{attribute addProperty BoxType "EL1259-0000-0018"}
{attribute addProperty Id "StatusAT %I*Status_8577222D3241InputsAT %I*Inputs_8B7B380018623.2533Input_event_timeAT %I*ARRAY[0 ..9] OF UDINT320400"}
{attribute addProperty CRC "3470487323"}
{attribute addProperty SizeInBites "538"}
{attribute addProperty SizeInBytes "67.25"}
TYPE MTI_Inputs_10x_Channel_28B0DBFB :
STRUCT
	{attribute addProperty Name "Status"}
	Status AT %I* : Status_8577222D;
	{attribute addProperty Name "Inputs"}
	Inputs AT %I* : Inputs_8B7B3800;
	{attribute addProperty Name "Input_event_time"}
	Input_event_time AT %I* : ARRAY[0 ..9] OF UDINT;
END_STRUCT
END_TYPE

(* stored: Version 1.2.0.0, ProductVersion 3.1.4024.9
   DUT MTI_Inputs_10x_Channel_28B0DBFB: Id {5dfae02d-b1f9-4b1b-9c40-a15231e0eb93} *)
